Staubli VAL3: onF4Event.pgx

program onF4Event()
  local point l_pPoint
begin
  // look if the bButton is enable
  if bButton[3]
    // get the tool
    call tcp:getTool(tTool,saveData:nFrameTool)
    l_pPoint=here(tTool,world)
    l_pPoint.trsf=align(l_pPoint.trsf,fSetFrame.trsf)
    movej(l_pPoint,tTool,nom_speed)
    call use:timerDialog(" ALIGN.... ",1)
    watch(isEmpty() or isKeyPressed(255),3)
    if !isEmpty()
      resetMotion()
    endIf
    delay(2)
  endIf
end
